% RSLogix 500 project I2P-Job-18 Duncan_Sutton.RSS, saved by version 10.00.00.00 %
PROJECT "ML01A"    % processor: Bul.1763 MicroLogix 1100 Series B %

PROGRAM FILES
  LAD 2   6 rungs

DATA FILES
  O0 OUTPUT  4 elements
  I1 INPUT  6 elements
  S2 STATUS  66 elements
  B3 BINARY  1 elements
  T4 TIMER  1 elements
  C5 COUNTER  1 elements
  R6 CONTROL  1 elements
  N7 INTEGER  1 elements
  F8 FLOAT  1 elements

LADDER 2
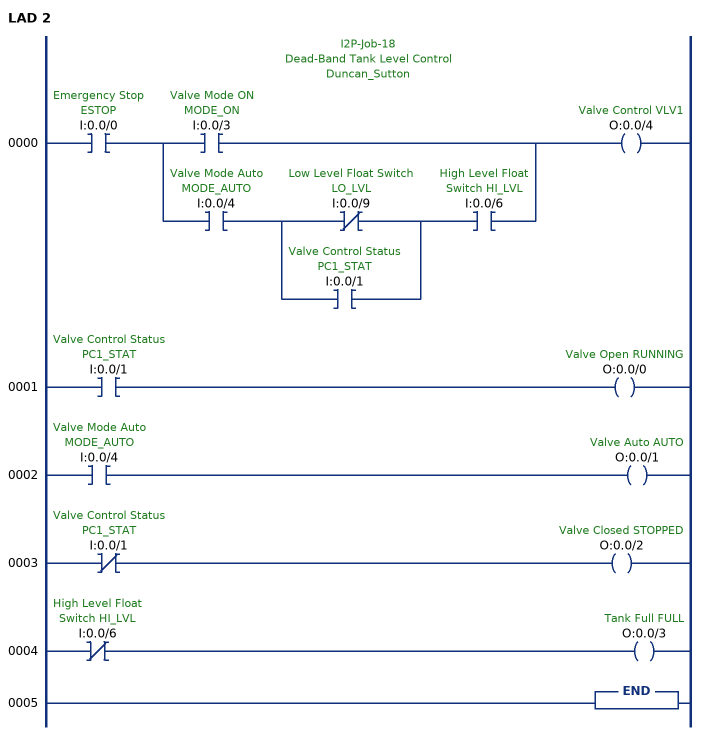
% Rung: 0 %
% I2P-Job-18
% Dead-Band Tank Level Control
% Duncan_Sutton %
SOR XIC I:0.0/0 BST XIC I:0.0/3 NXB XIC I:0.0/4 BST XIO I:0.0/9 NXB XIC I:0.0/1 BND XIC I:0.0/6 BND OTE O:0.0/4 EOR
%   I:0.0/0  ESTOP  "Emergency Stop" %
%   I:0.0/3  MODE_ON  "Valve Mode ON" %
%   I:0.0/4  MODE_AUTO  "Valve Mode Auto" %
%   I:0.0/9  LO_LVL  "Low Level Float Switch" %
%   I:0.0/1  PC1_STAT  "Valve Control Status" %
%   I:0.0/6  HI_LVL  "High Level Float Switch" %
%   O:0.0/4  VLV1  "Valve Control" %
% Rung: 1 %
SOR XIC I:0.0/1 OTE O:0.0/0 EOR
%   I:0.0/1  PC1_STAT  "Valve Control Status" %
%   O:0.0/0  RUNNING  "Valve Open" %
% Rung: 2 %
SOR XIC I:0.0/4 OTE O:0.0/1 EOR
%   I:0.0/4  MODE_AUTO  "Valve Mode Auto" %
%   O:0.0/1  AUTO  "Valve Auto" %
% Rung: 3 %
SOR XIO I:0.0/1 OTE O:0.0/2 EOR
%   I:0.0/1  PC1_STAT  "Valve Control Status" %
%   O:0.0/2  STOPPED  "Valve Closed" %
% Rung: 4 %
SOR XIO I:0.0/6 OTE O:0.0/3 EOR
%   I:0.0/6  HI_LVL  "High Level Float Switch" %
%   O:0.0/3  FULL  "Tank Full" %
% Rung: 5 %
SOR END EOR

OTHER DOCUMENTED ADDRESSES
  B3:0/0  B_ESTOP  "B_Estop"
  B3:0/1  B_FWD  "FWD Memory"
  B3:0/2  B_REV  "Reverse Memory"
  B3:0/3  LAST_FWD  "Memory Direction Foward"
  B3:0/4  LAST_REV  "Memory Direction Reverse"
  I:0.0/2  DIR_STAT  "Motor Direction Control Status"
  I:0.0/5  TMR_SEL
  I:0.0/7  START  "Motor Start"
  I:0.0/8  JOG  "JOG Motor"
  O:0.0/5  CR_2  "Direction Control Relay"
  T4:0.ACC/0  T4

DATA TABLE (non-zero values as saved)
DATA B3
% B3:0 % 0X0001
DATA T4
% .PRE .ACC %
% T4:0 % 32767 0
DATA C5
% .PRE .ACC %
% C5:0 % 16 0
